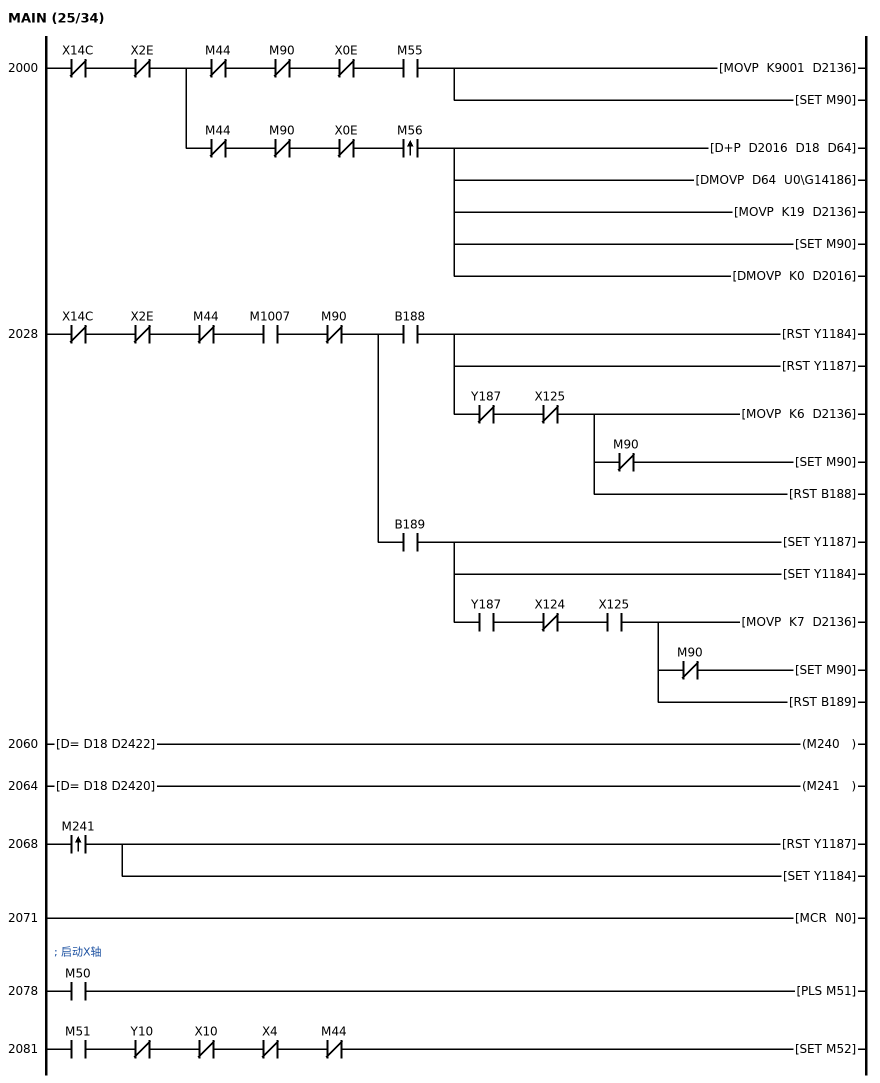
[picture p24: ladder of MAIN, rungs at steps 2000 to 2081]
2000  LDI     X14C
      ANI     X2E
      MPS
      ANI     M44
      ANI     M90
      ANI     X0E
      AND     M55
      MOVP    K9001 D2136
      SET     M90
      MPP
      ANI     M44
      ANI     M90
      ANI     X0E
      ANDP    M56
      D+P     D2016 D18 D64
      DMOVP   D64 U0\G14186
      MOVP    K19 D2136
      SET     M90
      DMOVP   K0 D2016
2028  LDI     X14C
      ANI     X2E
      ANI     M44
      AND     M1007
      ANI     M90
      MPS
      AND     B188
      RST     Y1184
      RST     Y1187
      ANI     Y187
      ANI     X125
      MOVP    K6 D2136
      MPS
      ANI     M90
      SET     M90
      MPP
      RST     B188
      MPP
      AND     B189
      SET     Y1187
      SET     Y1184
      AND     Y187
      ANI     X124
      AND     X125
      MOVP    K7 D2136
      MPS
      ANI     M90
      SET     M90
      MPP
      RST     B189
2060  LDD=    D18 D2422
      OUT     M240
2064  LDD=    D18 D2420
      OUT     M241
2068  LDP     M241
      RST     Y1187
      SET     Y1184
2071  MCR     N0
; 启动X轴
2078  LD      M50
      PLS     M51
2081  LD      M51
      ANI     Y10
      ANI     X10
      ANI     X4
      ANI     M44
      SET     M52
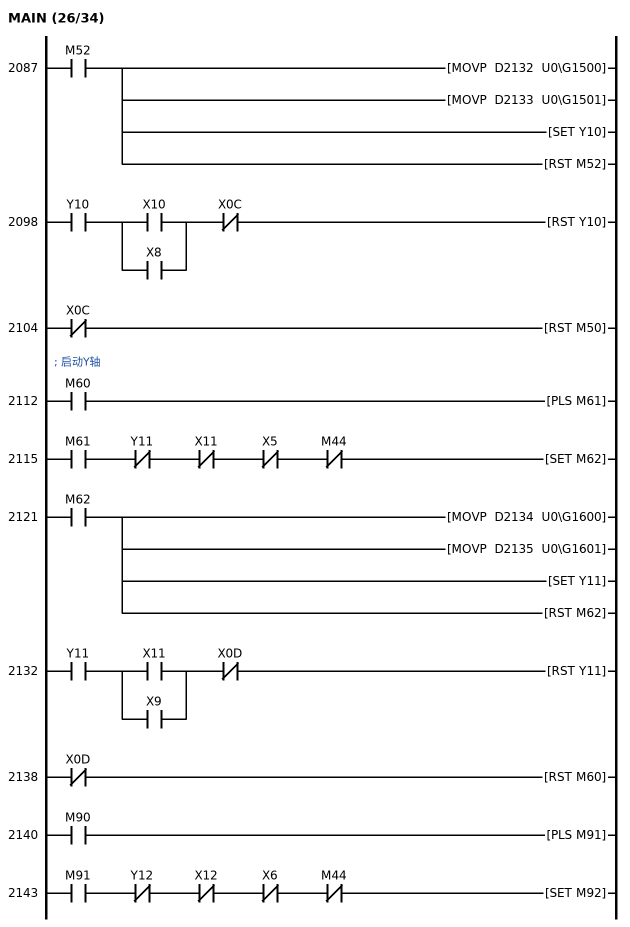
2087  LD      M52
      MOVP    D2132 U0\G1500
      MOVP    D2133 U0\G1501
      SET     Y10
      RST     M52
2098  LD      Y10
      LD      X10
      OR      X8
      ANB
      ANI     X0C
      RST     Y10
2104  LDI     X0C
      RST     M50
; 启动Y轴
2112  LD      M60
      PLS     M61
2115  LD      M61
      ANI     Y11
      ANI     X11
      ANI     X5
      ANI     M44
      SET     M62
2121  LD      M62
      MOVP    D2134 U0\G1600
      MOVP    D2135 U0\G1601
      SET     Y11
      RST     M62
2132  LD      Y11
      LD      X11
      OR      X9
      ANB
      ANI     X0D
      RST     Y11
2138  LDI     X0D
      RST     M60
2140  LD      M90
      PLS     M91
2143  LD      M91
      ANI     Y12
      ANI     X12
      ANI     X6
      ANI     M44
      SET     M92
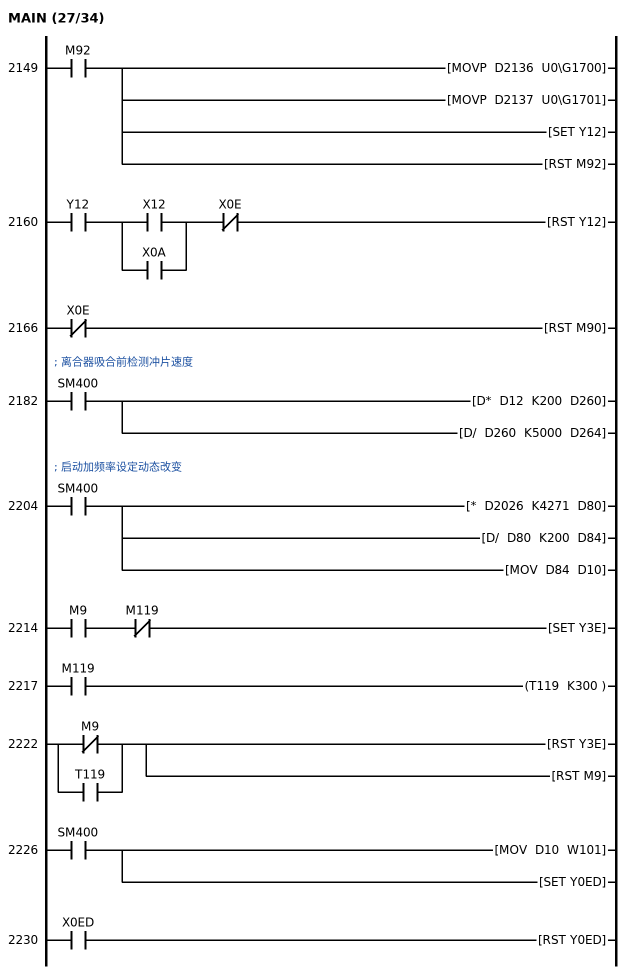
2149  LD      M92
      MOVP    D2136 U0\G1700
      MOVP    D2137 U0\G1701
      SET     Y12
      RST     M92
2160  LD      Y12
      LD      X12
      OR      X0A
      ANB
      ANI     X0E
      RST     Y12
2166  LDI     X0E
      RST     M90
; 离合器吸合前检测冲片速度
2182  LD      SM400
      D*      D12 K200 D260
      D/      D260 K5000 D264
; 启动加频率设定动态改变
2204  LD      SM400
      *       D2026 K4271 D80
      D/      D80 K200 D84
      MOV     D84 D10
2214  LD      M9
      ANI     M119
      SET     Y3E
2217  LD      M119
      OUT     T119 K300
2222  LDI     M9
      OR      T119
      RST     Y3E
      RST     M9
2226  LD      SM400
      MOV     D10 W101
      SET     Y0ED
2230  LD      X0ED
      RST     Y0ED
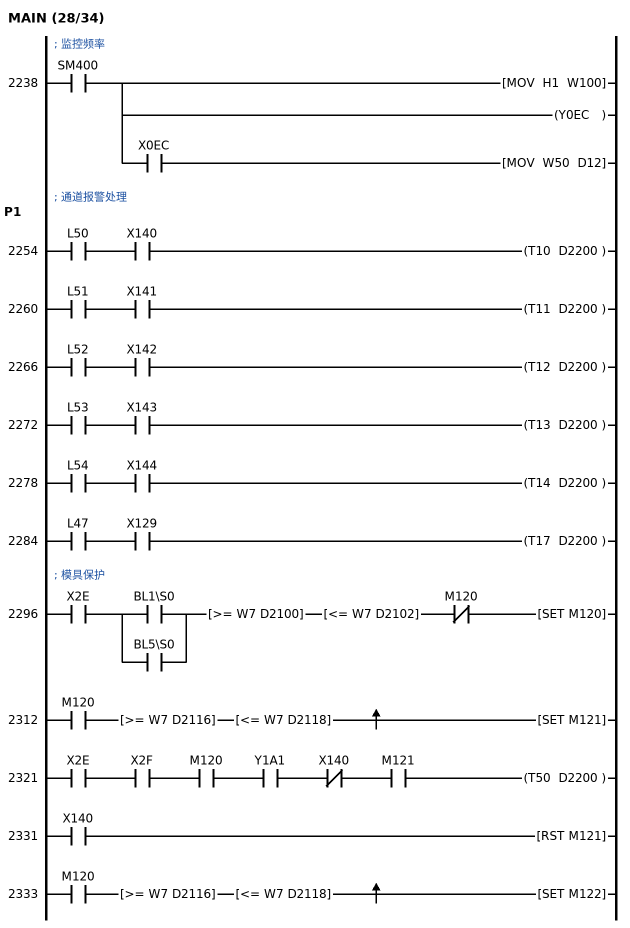
; 监控频率
2238  LD      SM400
      MOV     H1 W100
      OUT     Y0EC
      AND     X0EC
      MOV     W50 D12
; 通道报警处理
      P1
2254  LD      L50
      AND     X140
      OUTH    T10 D2200
2260  LD      L51
      AND     X141
      OUTH    T11 D2200
2266  LD      L52
      AND     X142
      OUTH    T12 D2200
2272  LD      L53
      AND     X143
      OUTH    T13 D2200
2278  LD      L54
      AND     X144
      OUTH    T14 D2200
2284  LD      L47
      AND     X129
      OUTH    T17 D2200
; 模具保护
2296  LD      X2E
      LD      BL1\S0
      OR      BL5\S0
      ANB
      AND>=   W7 D2100
      AND<=   W7 D2102
      ANI     M120
      SET     M120
2312  LD      M120
      AND>=   W7 D2116
      AND<=   W7 D2118
      MEP
      SET     M121
2321  LD      X2E
      AND     X2F
      AND     M120
      AND     Y1A1
      ANI     X140
      AND     M121
      OUTH    T50 D2200
2331  LD      X140
      RST     M121
2333  LD      M120
      AND>=   W7 D2116
      AND<=   W7 D2118
      MEP
      SET     M122
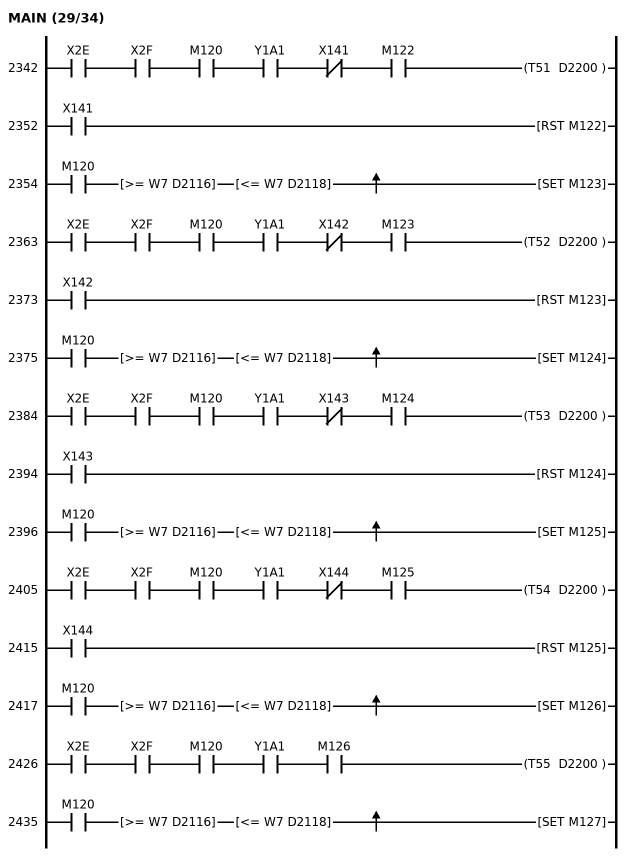
2342  LD      X2E
      AND     X2F
      AND     M120
      AND     Y1A1
      ANI     X141
      AND     M122
      OUTH    T51 D2200
2352  LD      X141
      RST     M122
2354  LD      M120
      AND>=   W7 D2116
      AND<=   W7 D2118
      MEP
      SET     M123
2363  LD      X2E
      AND     X2F
      AND     M120
      AND     Y1A1
      ANI     X142
      AND     M123
      OUTH    T52 D2200
2373  LD      X142
      RST     M123
2375  LD      M120
      AND>=   W7 D2116
      AND<=   W7 D2118
      MEP
      SET     M124
2384  LD      X2E
      AND     X2F
      AND     M120
      AND     Y1A1
      ANI     X143
      AND     M124
      OUTH    T53 D2200
2394  LD      X143
      RST     M124
2396  LD      M120
      AND>=   W7 D2116
      AND<=   W7 D2118
      MEP
      SET     M125
2405  LD      X2E
      AND     X2F
      AND     M120
      AND     Y1A1
      ANI     X144
      AND     M125
      OUTH    T54 D2200
2415  LD      X144
      RST     M125
2417  LD      M120
      AND>=   W7 D2116
      AND<=   W7 D2118
      MEP
      SET     M126
2426  LD      X2E
      AND     X2F
      AND     M120
      AND     Y1A1
      AND     M126
      OUTH    T55 D2200
2435  LD      M120
      AND>=   W7 D2116
      AND<=   W7 D2118
      MEP
      SET     M127
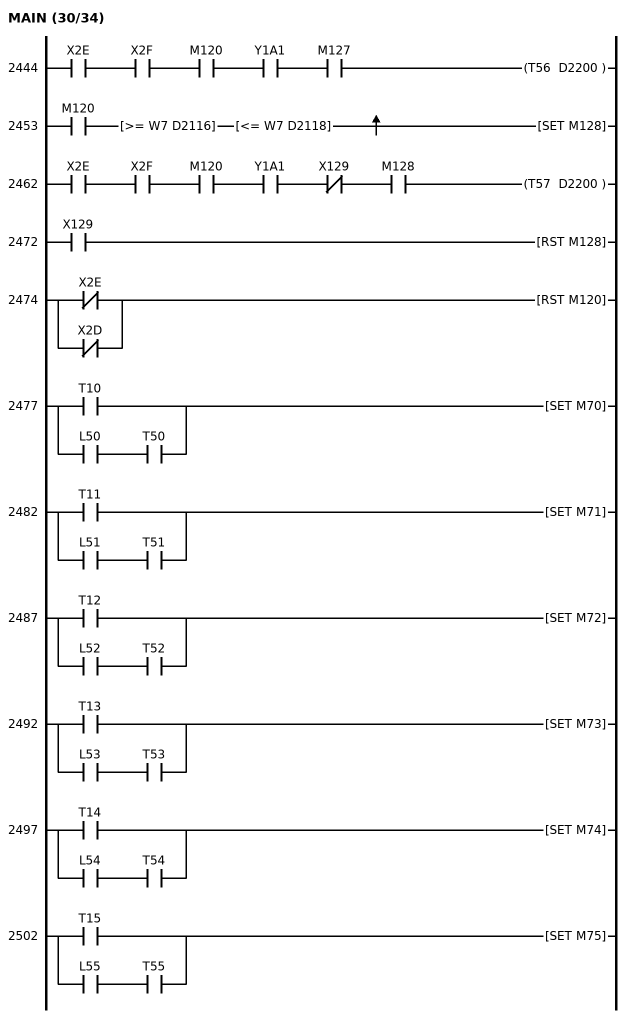
2444  LD      X2E
      AND     X2F
      AND     M120
      AND     Y1A1
      AND     M127
      OUTH    T56 D2200
2453  LD      M120
      AND>=   W7 D2116
      AND<=   W7 D2118
      MEP
      SET     M128
2462  LD      X2E
      AND     X2F
      AND     M120
      AND     Y1A1
      ANI     X129
      AND     M128
      OUTH    T57 D2200
2472  LD      X129
      RST     M128
2474  LDI     X2E
      ORI     X2D
      RST     M120
2477  LD      T10
      LD      L50
      AND     T50
      ORB
      SET     M70
2482  LD      T11
      LD      L51
      AND     T51
      ORB
      SET     M71
2487  LD      T12
      LD      L52
      AND     T52
      ORB
      SET     M72
2492  LD      T13
      LD      L53
      AND     T53
      ORB
      SET     M73
2497  LD      T14
      LD      L54
      AND     T54
      ORB
      SET     M74
2502  LD      T15
      LD      L55
      AND     T55
      ORB
      SET     M75
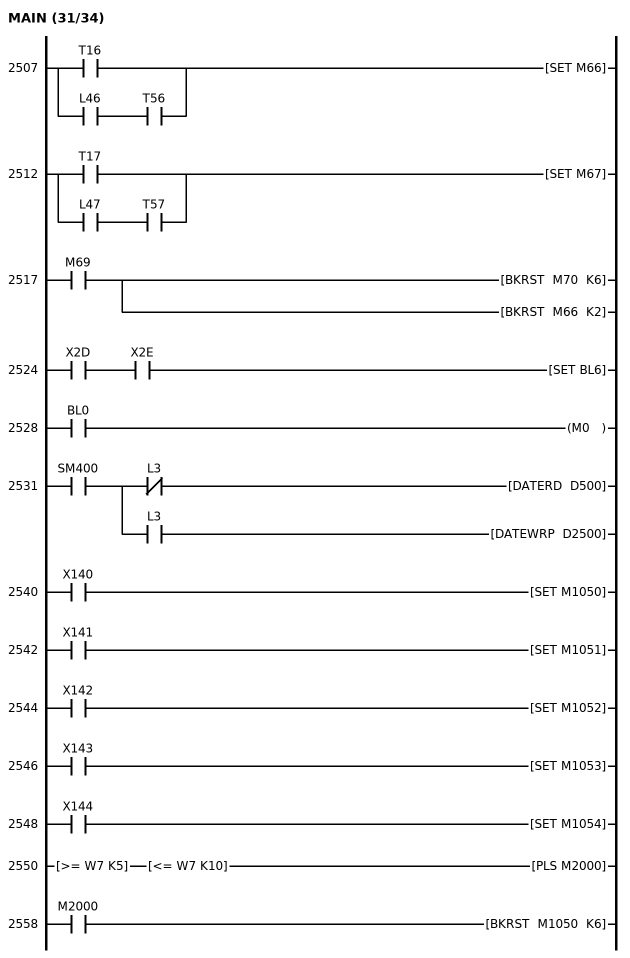
2507  LD      T16
      LD      L46
      AND     T56
      ORB
      SET     M66
2512  LD      T17
      LD      L47
      AND     T57
      ORB
      SET     M67
2517  LD      M69
      BKRST   M70 K6
      BKRST   M66 K2
2524  LD      X2D
      AND     X2E
      SET     BL6
2528  LD      BL0
      OUT     M0
2531  LD      SM400
      MPS
      ANI     L3
      DATERD  D500
      MPP
      AND     L3
      DATEWRP D2500
2540  LD      X140
      SET     M1050
2542  LD      X141
      SET     M1051
2544  LD      X142
      SET     M1052
2546  LD      X143
      SET     M1053
2548  LD      X144
      SET     M1054
2550  LD>=    W7 K5
      AND<=   W7 K10
      PLS     M2000
2558  LD      M2000
      BKRST   M1050 K6
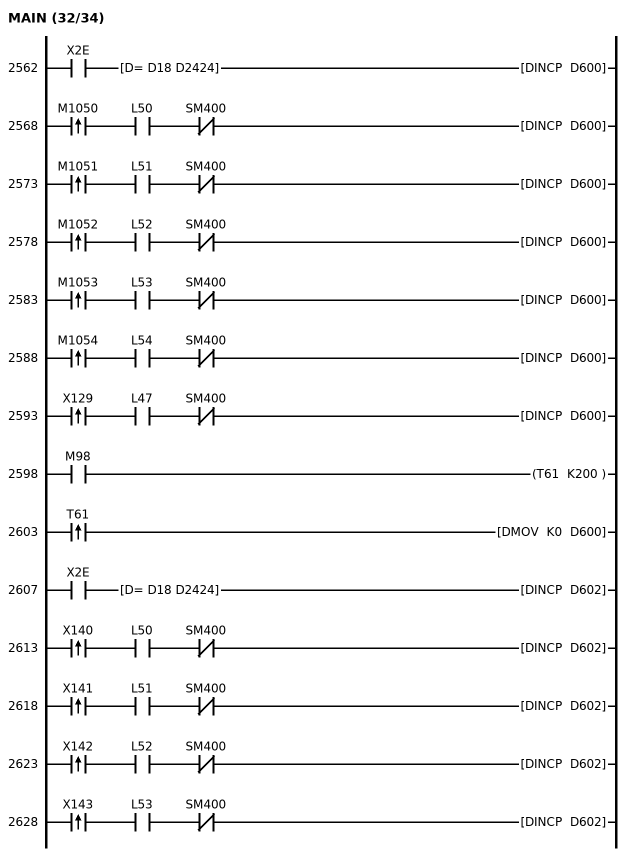
2562  LD      X2E
      ANDD=   D18 D2424
      DINCP   D600
2568  LDP     M1050
      AND     L50
      ANI     SM400
      DINCP   D600
2573  LDP     M1051
      AND     L51
      ANI     SM400
      DINCP   D600
2578  LDP     M1052
      AND     L52
      ANI     SM400
      DINCP   D600
2583  LDP     M1053
      AND     L53
      ANI     SM400
      DINCP   D600
2588  LDP     M1054
      AND     L54
      ANI     SM400
      DINCP   D600
2593  LDP     X129
      AND     L47
      ANI     SM400
      DINCP   D600
2598  LD      M98
      OUT     T61 K200
2603  LDP     T61
      DMOV    K0 D600
2607  LD      X2E
      ANDD=   D18 D2424
      DINCP   D602
2613  LDP     X140
      AND     L50
      ANI     SM400
      DINCP   D602
2618  LDP     X141
      AND     L51
      ANI     SM400
      DINCP   D602
2623  LDP     X142
      AND     L52
      ANI     SM400
      DINCP   D602
2628  LDP     X143
      AND     L53
      ANI     SM400
      DINCP   D602
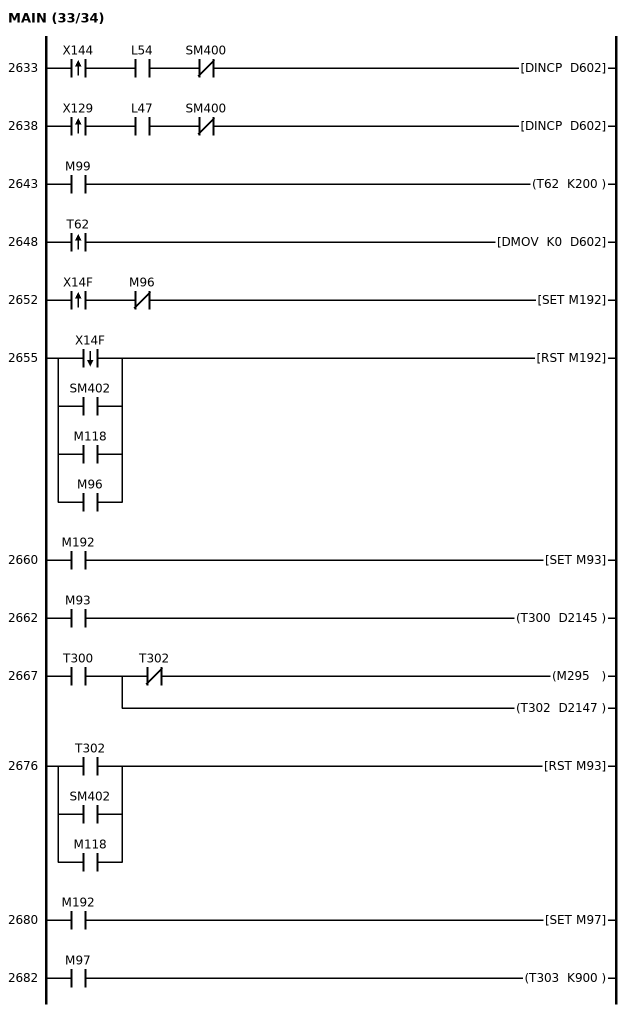
2633  LDP     X144
      AND     L54
      ANI     SM400
      DINCP   D602
2638  LDP     X129
      AND     L47
      ANI     SM400
      DINCP   D602
2643  LD      M99
      OUT     T62 K200
2648  LDP     T62
      DMOV    K0 D602
2652  LDP     X14F
      ANI     M96
      SET     M192
2655  LDF     X14F
      OR      SM402
      OR      M118
      OR      M96
      RST     M192
2660  LD      M192
      SET     M93
2662  LD      M93
      OUTH    T300 D2145
2667  LD      T300
      MPS
      ANI     T302
      OUT     M295
      MPP
      OUTH    T302 D2147
2676  LD      T302
      OR      SM402
      OR      M118
      RST     M93
2680  LD      M192
      SET     M97
2682  LD      M97
      OUT     T303 K900
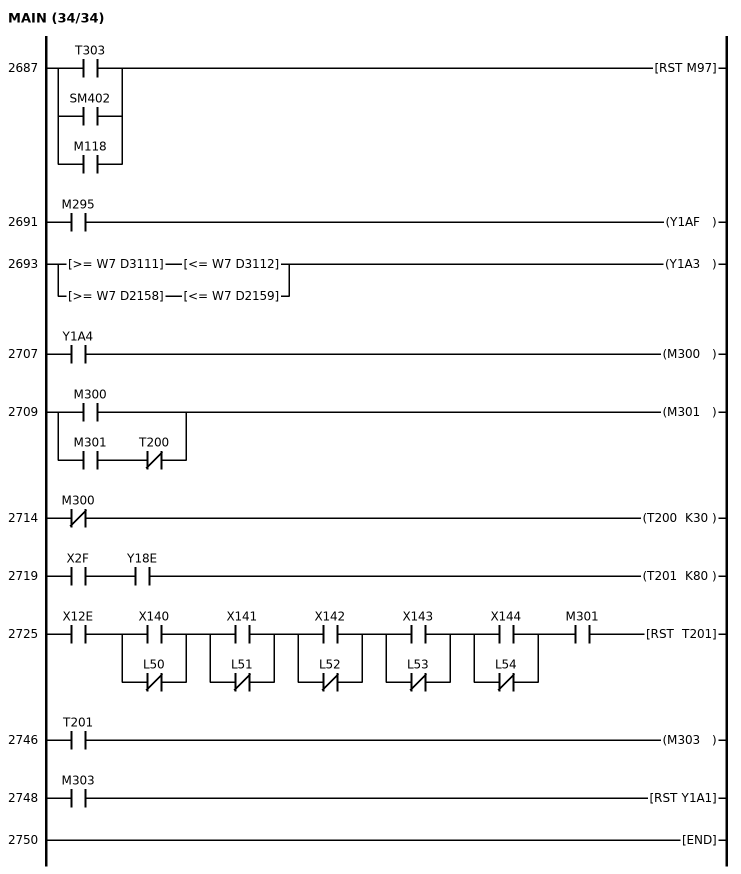
2687  LD      T303
      OR      SM402
      OR      M118
      RST     M97
2691  LD      M295
      OUT     Y1AF
2693  LD>=    W7 D3111
      AND<=   W7 D3112
      LD>=    W7 D2158
      AND<=   W7 D2159
      ORB
      OUT     Y1A3
2707  LD      Y1A4
      OUT     M300
2709  LD      M300
      LD      M301
      ANI     T200
      ORB
      OUT     M301
2714  LDI     M300
      OUT     T200 K30
2719  LD      X2F
      AND     Y18E
      OUT     T201 K80
2725  LD      X12E
      LD      X140
      ORI     L50
      ANB
      LD      X141
      ORI     L51
      ANB
      LD      X142
      ORI     L52
      ANB
      LD      X143
      ORI     L53
      ANB
      LD      X144
      ORI     L54
      ANB
      AND     M301
      RST     T201
2746  LD      T201
      OUT     M303
2748  LD      M303
      RST     Y1A1
2750  END
END_PROGRAM
